TYPE ST_ReturnStructure :
STRUCT
	Done	: BOOL;
	Active	: BOOL;
	Busy	: BOOL;
	Aborted	: BOOL;
	Error	: BOOL;
	ErrorId	: UDINT;
END_STRUCT
END_TYPE

(* stored: Version 1.1.0.1, ProductVersion 3.1.4026.12
   DUT ST_ReturnStructure: Id {e71565bb-ab22-0e36-3a34-064ddeb2e9cf} *)
